TYPE BufferTC_DivertComm :
STRUCT
	NeedEmpties: BOOL;
	NeedFullPriorityNormal: BOOL;
	NeedFullPriorityHigh: BOOL;
END_STRUCT
END_TYPE

(* stored: Version 1.1.0.1, ProductVersion 3.1.4024.6
   DUT BufferTC_DivertComm: Id {e59977d2-43cf-45cf-8c71-0747421168c3} *)
